(* PLC project safeApp1, BrAutomation SafeDESIGNER  5.16.0.0 *)
(* stored: companyURL http://www.br-automation.com, creationDateTime Thu Apr 28 11:09:09 2022 *)

PROGRAM Main

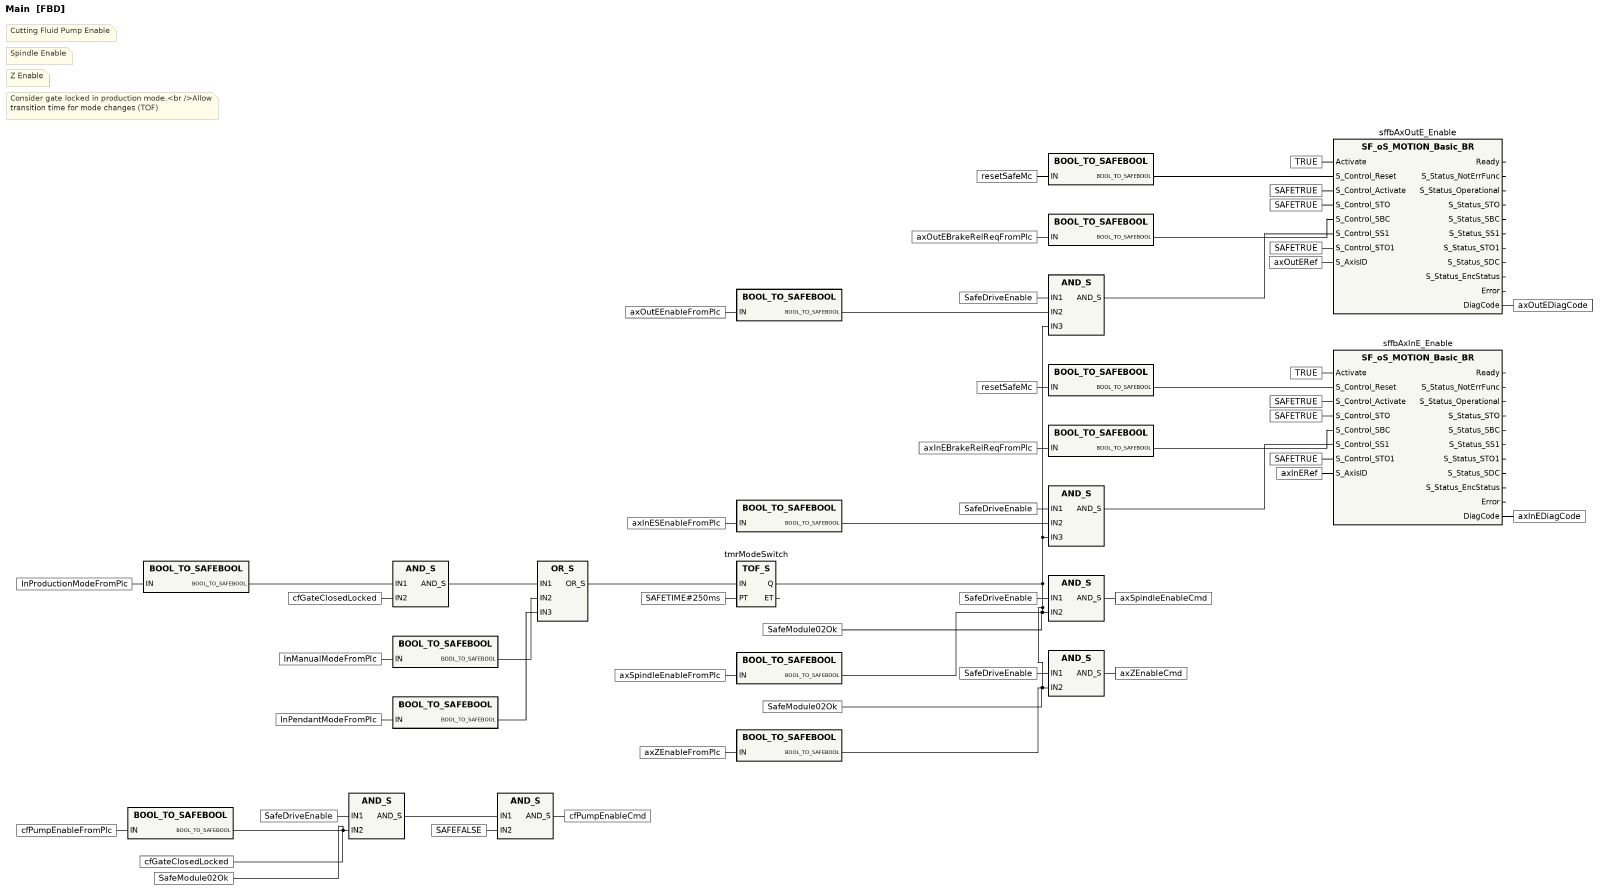
(* FBD diagram, written out as Structured Text *)
(* Consider gate locked in production mode.<br />Allow transition time for mode changes (TOF) *)
tmrModeSwitch(IN := OR_S(AND_S(BOOL_TO_SAFEBOOL(InProductionModeFromPlc), cfGateClosedLocked), BOOL_TO_SAFEBOOL(InManualModeFromPlc), BOOL_TO_SAFEBOOL(InPendantModeFromPlc)), PT := SAFETIME#250ms);
sffbAxOutE_Enable(Activate := TRUE, S_Control_Reset := BOOL_TO_SAFEBOOL(resetSafeMc), S_Control_Activate := SAFETRUE, S_Control_STO := SAFETRUE, S_Control_SBC := BOOL_TO_SAFEBOOL(axOutEBrakeRelReqFromPlc), S_Control_SS1 := AND_S(SafeDriveEnable, BOOL_TO_SAFEBOOL(axOutEEnableFromPlc), tmrModeSwitch.Q), S_Control_STO1 := SAFETRUE, S_AxisID := axOutERef);
axOutEDiagCode := sffbAxOutE_Enable.DiagCode;
sffbAxInE_Enable(Activate := TRUE, S_Control_Reset := BOOL_TO_SAFEBOOL(resetSafeMc), S_Control_Activate := SAFETRUE, S_Control_STO := SAFETRUE, S_Control_SBC := BOOL_TO_SAFEBOOL(axInEBrakeRelReqFromPlc), S_Control_SS1 := AND_S(SafeDriveEnable, BOOL_TO_SAFEBOOL(axInESEnableFromPlc), tmrModeSwitch.Q), S_Control_STO1 := SAFETRUE, S_AxisID := axInERef);
axInEDiagCode := sffbAxInE_Enable.DiagCode;
(* Spindle Enable *)
axSpindleEnableCmd := AND_S(SafeDriveEnable, BOOL_TO_SAFEBOOL(axSpindleEnableFromPlc), tmrModeSwitch.Q, SafeModule02Ok);
(* Z Enable *)
axZEnableCmd := AND_S(SafeDriveEnable, BOOL_TO_SAFEBOOL(axZEnableFromPlc), tmrModeSwitch.Q, SafeModule02Ok);
(* Cutting Fluid Pump Enable *)
cfPumpEnableCmd := AND_S(AND_S(SafeDriveEnable, BOOL_TO_SAFEBOOL(cfPumpEnableFromPlc), cfGateClosedLocked, SafeModule02Ok), SAFEFALSE);
END_PROGRAM
